FUNCTION_BLOCK FB_HeatExchanger1 EXTENDS FB_SystemContinous
VAR_INPUT
END_VAR
VAR_OUTPUT
END_VAR
VAR
END_VAR

(*
- implementierung ähnlich zu wärmetauscher system bei hvfa speichern
- bestehend aus 2 Magna 3 pumpen (PU315, PU215)
- disrcete valve SV315
- mixing valve RV215
- heat counter WMZ215

Logik:
- RampUp: SV und RV öffnen
- Operational: PUs anschalten
- Working: RV regelt auf Vorlauftemepratur an PWT1
- RampDown: Umgekehrte Reihenfolge

- errorCheck: Prüfe auf pumpenerror, falls SV315 Stellugnsrückmeldung hat (in aktuellem bei Verknüpfungen prüfen), dann prüfen ob pumpe gegen geschlossenes Ventil pumpt
*)

END_FUNCTION_BLOCK

(* stored: Version 1.1.0.1, ProductVersion 3.1.4024.10
   POU FB_HeatExchanger1: Id {bca56c6b-1b09-4f57-a186-5b7562770c5b}, SpecialFunc None *)
